// TwinCAT 3 PLC project MoottoriSylinteri
// ProgramVersion: 3.1.4023.0
// libraries:
//   Tc2_Standard, * (Beckhoff Automation GmbH)
//   Tc2_System, * (Beckhoff Automation GmbH)
//   Tc3_Module, * (Beckhoff Automation GmbH)
//   VisuSymbols,3.5.10.0,System
// project tree:
//   / GlobalTextList.TcGTLO, PlcTask.TcTTO, Visualization Manager.TcVMO (not stored)
//   POUs/ MAIN.TcPOU
//   VISUs/ Visualization.TcVIS
// real-time tasks:
//   TASK PlcTask: cycle T#10ms, priority 20, ADS port 350

CONFIGURATION MoottoriSylinteri
    RESOURCE PLC ON TwinCAT3
        TASK PlcTask(INTERVAL := T#10ms, PRIORITY := 20);
        PROGRAM MAIN WITH PlcTask : MAIN;
    END_RESOURCE
END_CONFIGURATION

// ---- POUs/MAIN.TcPOU
PROGRAM MAIN
VAR
	start : BOOL;
	stop : BOOL;
	lamppu : BOOL;
	ton3: TON;
	step : INT;
END_VAR

VAR_INPUT
	iCyl1minus AT %IX0.0: BOOL;
	iCyl1plus AT %IX0.1: BOOL;
	iCyl2minus AT %IX0.3: BOOL;
	iCyl2plus AT %IX0.4: BOOL;
	iCyl3minus AT %IX1.0: BOOL;
	iCyl3plus AT %IX1.1: BOOL;
	iCyl4minus AT %IX1.3: BOOL;
	iCyl4plus AT %IX1.4: BOOL;
	iMot1running AT %IX0.2: BOOL;
	iMot2running AT %IX0.5: BOOL;
	iMot3running AT %IX1.2: BOOL;
	iMot4running AT %IX1.5: BOOL;
END_VAR

VAR_OUTPUT
	qCyl1toMinus AT %QX0.0: BOOL;
	qCyl1toPlus AT %QX0.1: BOOL;
	qCyl2toMinus AT %QX0.3: BOOL;
	qCyl2toPlus AT %QX0.4: BOOL;
	qCyl3toMinus AT %QX1.0: BOOL;
	qCyl3toPlus AT %QX1.1: BOOL;
	qCyl4toMinus AT %QX1.3: BOOL;
	qCyl4toPlus AT %QX1.4: BOOL;
	qMot1start AT %QX0.2: BOOL;
	qMot2start AT %QX0.5: BOOL;
	qMot3start AT %QX1.2: BOOL;
	qMot4start AT %QX1.5: BOOL;
END_VAR

// nollataan lähdöt joka kierroksen alussa
qMot1start := FALSE;
qCyl1toMinus := FALSE;
qCyl1toPlus := FALSE;
lamppu := FALSE;

IF stop THEN
	step := 0;
END_IF

CASE step OF
	0: // odotus
		IF start AND NOT iMot1running AND iCyl1minus THEN
			step := 10;
		END_IF
	
	10: // moottori käynnistyy
		qMot1start := TRUE;
		IF iMot1running THEN
			step := 20;
		END_IF
	20: // sylinteri oikealle
		qMot1start := TRUE;
		qCyl1toPlus := TRUE;
		IF iCyl1plus THEN
			step := 30;
		END_IF
	30: // sylinteri vasemmalle
		qMot1start := TRUE;
		qCyl1toMinus := TRUE;
		IF iCyl1minus THEN
			step := 40;
		END_IF
	40: // moottori sammuu
		IF NOT iMot1running THEN
			step := 50;
		END_IF
	50: lamppu := TRUE;
	
END_CASE

END_PROGRAM

// ---- VISUs/Visualization.TcVIS
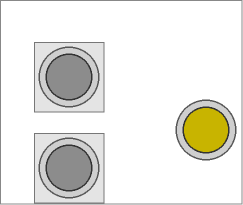
VISUALIZATION Visualization  // 243x205
    Lamp1 (171,95 70x70), variable: MAIN.lamppu, style: Lamp-Lamp1-Yellow
    PushSwitch (34,42 70x70), variable: MAIN.start, behaviour: TAP, style: Switch-PushSwitch-Gray
    PushSwitch (34,133 70x70), variable: MAIN.stop, behaviour: TAP, style: Switch-PushSwitch-Gray
END_VISUALIZATION
